{attribute 'GeneratedUsingTerminal: EK1122-0000-0018'}
{attribute addProperty BoxType "EK1122-0000-0018"}
{attribute addProperty Id "Beckhoff_EL99xxsub_EK1100EK1100_1FC0878B2"}
{attribute addProperty CRC "1792639607"}
{attribute addProperty Size "2"}
TYPE Beckhoff_EL99xxEK1122_6AD98277 EXTENDS EK1122_1FC0878B :
STRUCT
	{attribute addProperty Name "Beckhoff_EL99xxsub_EK1100"}
	{attribute addProperty PreviousPort "Beckhoff EL99xxEK1122 : D"}
	Beckhoff_EL99xxsub_EK1100 : EK1100_1FC0878B;
END_STRUCT
END_TYPE

(* stored: Version 1.2.0.0, ProductVersion 3.1.4024.9
   DUT Beckhoff_EL99xxEK1122_6AD98277: Id {09b8f187-f952-4d57-b588-887c0bbaf56d} *)
